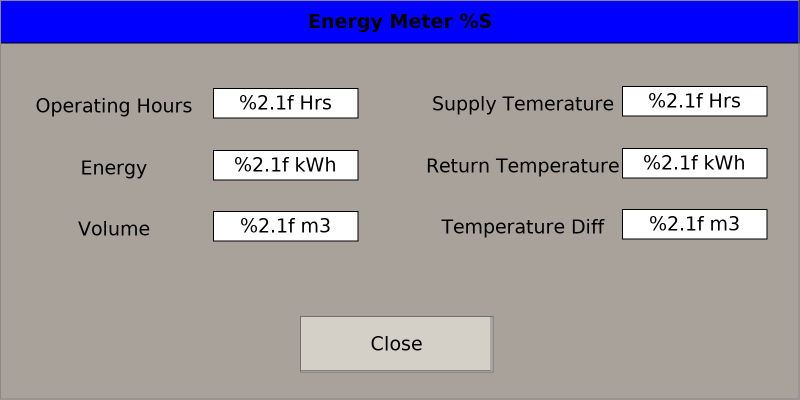
VISUALIZATION Dialog_EnergyMeter  // 800x400
VAR_IN_OUT
	sHeader : STRING;
	fOperHours: REAL;
	fEnergy: REAL;
	fVolume: REAL;
	fSupply_Temp:REAL;
	fReturn_Temp : REAL;
	fReturn_Diff: REAL;

END_VAR
    Rectangle (0,0 800x43), "Energy Meter %S", text variable: sHeader
    Label (19,92 190x28), "Operating Hours"
    Label (19,154 190x28), "Energy"
    Label (19,215 190x28), "Volume"
    Rectangle (213,88 145x30), "%2.1f Hrs", text variable: fOperHours
    Rectangle (213,150 145x30), "%2.1f kWh", text variable: fEnergy
    Rectangle (213,211 145x30), "%2.1f m3", text variable: fVolume
    Label (428,90 190x28), "Supply Temerature"
    Label (428,152 190x28), "Return Temperature"
    Label (428,213 190x28), "Temperature Diff"
    Rectangle (622,86 145x30), "%2.1f Hrs", text variable: fSupply_Temp
    Rectangle (622,148 145x30), "%2.1f kWh", text variable: fReturn_Temp
    Rectangle (622,209 145x30), "%2.1f m3", text variable: fReturn_Diff
    Button (300,316 193x56), "Close"
END_VISUALIZATION

(* stored: Version 1.1.0.1, ProductVersion 3.1.4024.12
   Visu Dialog_EnergyMeter: Id {c5568d72-8a16-4159-8009-208bbe4aea83} *)
